// TIA Portal V16 export
// export: Created 2023-03-29T11:03:18.5834771Z, ExportSetting WithDefaults, DisplayName Totally Integrated Automation Portal, DisplayVersion V16 Update 6, DisplayName TIA Portal Version Control Interface, DisplayVersion V16 Update 2, DisplayName TIA Portal Openness, DisplayVersion V16 Update 6, DisplayName STEP 7 Professional, DisplayVersion V16 Update 6, DisplayName STEP 7 Safety, DisplayVersion V16, DisplayName WinCC Advanced, DisplayVersion V16 Update 6
ORGANIZATION_BLOCK "Cyclic interrupt_ModbusTCP_wysyłanie"   // OB30, LAD, CyclicInterrupt
{ S7_Optimized_Access := 'TRUE' }
VERSION : 0.1
// stored: AutoNumber true, IsIECCheckEnabled false, SetENOAutomatically false
   VAR_INPUT
      Initial_Call : Bool;   // Initial call of this OB
      Event_Count : Int;   // Events discarded
   END_VAR
BEGIN

REGION Network 1: Odczyt poziomów w zbiornku
END_REGION

REGION Network 2 (SCL): Odczyt poziomów w zbiornku
   "AI_poziom_zbiornik_1" := "IW68";
   "AI_poziom_zbiornik_2" := "IW70";
   "AI_poziom_zbiornik_3" := "IW72";
   "AI_poziom_zbiornik_4" := "IW74";

   "AI_położenie_Z10" := "IW78";
END_REGION

REGION Network 3 (SCL): Ciśnienie magistrala

   IF "IW76":P > 0.2 THEN // czy nie uszkodzone rury
     IF "IW76":P < 27651 THEN // przerwana pętla prądowa
       // to przekazanie wartości
       "AI_ciśnienie_B5" := "IW76":P;
       ;
     ELSE
       "AI_ciśnienie_B5" := 32767;
       ;
     END_IF;

     ;
   END_IF;
END_REGION

REGION Network 4 (SCL): Położenie zasuwy Z10
   // Odczyt w FC5
END_REGION
END_ORGANIZATION_BLOCK
